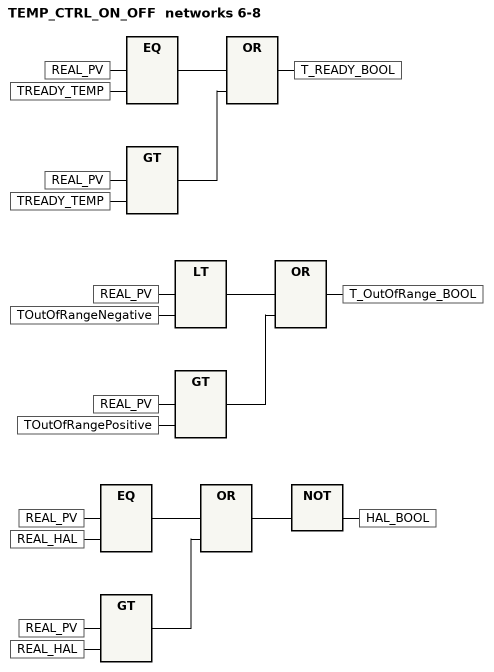
[picture p96: TEMP_CTRL_ON_OFF (FBD) networks 6-8]
_FBD_ (* Function Block Diagram *)
NETWORK 1
	DIV(INT_TO_REAL(TEMP_PV), 10) => REAL_PV
NETWORK 2
	T1:TON(IN: NOT ALWAYS_OFF, PT: T#100ms) => ALWAYS_ON_BOOL
NETWORK 3
	SUB(REAL_SV, REAL_T_READY) => TREADY_TEMP
NETWORK 4
	SUB(REAL_SV, REAL_HYS) => HYS_TEMP
NETWORK 5
	RS1:RS(SET: OR(AND(PLS1:R_TRIG(CLK: ALWAYS_ON_BOOL), LT(REAL_PV, REAL_SV)), OR(EQ(REAL_PV, HYS_TEMP), LT(REAL_PV, HYS_TEMP))), RESET1: OR(OR(EQ(REAL_PV, REAL_SV), GT(REAL_PV, REAL_SV)), NOT HAL_BOOL)) => OUT_BOOL
NETWORK 6
	OR(EQ(REAL_PV, TREADY_TEMP), GT(REAL_PV, TREADY_TEMP)) => T_READY_BOOL
NETWORK 7
	OR(LT(REAL_PV, TOutOfRangeNegative), GT(REAL_PV, TOutOfRangePositive)) => T_OutOfRange_BOOL
NETWORK 8
	NOT OR(EQ(REAL_PV, REAL_HAL), GT(REAL_PV, REAL_HAL)) => HAL_BOOL
_END_FBD_
(* the same logic as Structured Text *)
(* Network 1 *)
REAL_PV := INT_TO_REAL(TEMP_PV) / 10;
(* Network 2 *)
T1(IN := NOT ALWAYS_OFF, PT := T#100ms);
ALWAYS_ON_BOOL := T1.Q;
(* Network 3 *)
TREADY_TEMP := REAL_SV - REAL_T_READY;
(* Network 4 *)
HYS_TEMP := REAL_SV - REAL_HYS;
(* Network 5 *)
PLS1(CLK := ALWAYS_ON_BOOL);
RS1(SET := (PLS1.Q AND (REAL_PV < REAL_SV)) OR ((REAL_PV = HYS_TEMP) OR (REAL_PV < HYS_TEMP)), RESET1 := ((REAL_PV = REAL_SV) OR (REAL_PV > REAL_SV)) OR NOT HAL_BOOL);
OUT_BOOL := RS1.Q1;
(* Network 6 *)
T_READY_BOOL := (REAL_PV = TREADY_TEMP) OR (REAL_PV > TREADY_TEMP);
(* Network 7 *)
T_OutOfRange_BOOL := (REAL_PV < TOutOfRangeNegative) OR (REAL_PV > TOutOfRangePositive);
(* Network 8 *)
HAL_BOOL := NOT ((REAL_PV = REAL_HAL) OR (REAL_PV > REAL_HAL));
END_FUNCTION_BLOCK

(* POU TIMER_ALARM, LD *)
FUNCTION_BLOCK TIMER_ALARM
VAR_INPUT
	BOOL_SIGNAL_IN: BOOL;
	BOOL_ALMRST_PB: BOOL;
	BOOL_BZRST_PB: BOOL;
	INT_PV: INT;

END_VAR

VAR_OUTPUT
	ALM_MSG_BOOL: BOOL;
	BZ_OUT_BOOL: BOOL;
	EV_INT: INT;
END_VAR

VAR
	T1: TON;
	M0: BOOL;
	M1: BOOL;
	D200: TIME;
	D202: INT;
END_VAR
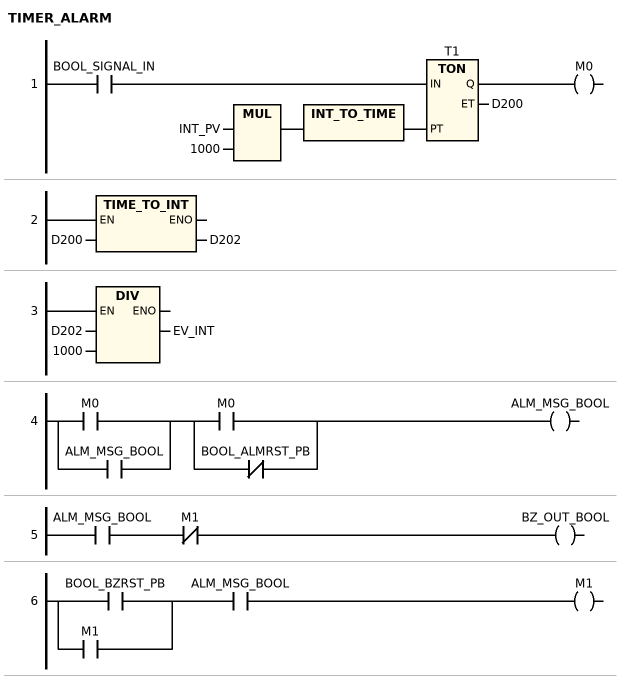
_LD_ (* Ladder Diagram *)
NETWORK 1
	[BOOL_SIGNAL_IN] - T1:TON(IN: *, PT: INT_TO_TIME(MUL(INT_PV, 1000)), ET => D200) --- (M0)
NETWORK 2
	*
		EN --- TIME_TO_INT(D200) => D202
NETWORK 3
	*
		EN --- DIV(D202, 1000) => EV_INT
NETWORK 4
	{ [M0] | [ALM_MSG_BOOL] } - { [M0] | [/BOOL_ALMRST_PB] } --- (ALM_MSG_BOOL)
NETWORK 5
	[ALM_MSG_BOOL] - [/M1] --- (BZ_OUT_BOOL)
NETWORK 6
	{ [BOOL_BZRST_PB] | [M1] } - [ALM_MSG_BOOL] --- (M1)
_END_LD_
(* the same logic as Structured Text *)
(* Network 1 *)
T1(IN := BOOL_SIGNAL_IN, PT := INT_TO_TIME(INT_PV * 1000));
D200 := T1.ET;
M0 := T1.Q;
(* Network 2 *)
D202 := TIME_TO_INT(D200);
(* Network 3 *)
EV_INT := D202 / 1000;
(* Network 4 *)
ALM_MSG_BOOL := (M0 OR ALM_MSG_BOOL) AND (M0 OR NOT BOOL_ALMRST_PB);
(* Network 5 *)
BZ_OUT_BOOL := ALM_MSG_BOOL AND NOT M1;
(* Network 6 *)
M1 := (BOOL_BZRST_PB OR M1) AND ALM_MSG_BOOL;
END_FUNCTION_BLOCK

(* POU TOWER_LIGHT, LD *)
FUNCTION_BLOCK TOWER_LIGHT
VAR_INPUT

	bAlarmOccur : BOOL;
	bMainOnOff : BOOL;
	bAutoStart : BOOL;
	bAutoProgress : BOOL;
	bAutoCycleStop: BOOL;
	bManualMode : BOOL;



END_VAR
VAR_OUTPUT
	bTowerLightRED : BOOL;
	bTowerLightYELLOW : BOOL;
	bTowerLightGREEN : BOOL;

END_VAR
VAR

	AlwaysOn : BOOL := TRUE;

	T1: TON;
	T2: TON;
END_VAR
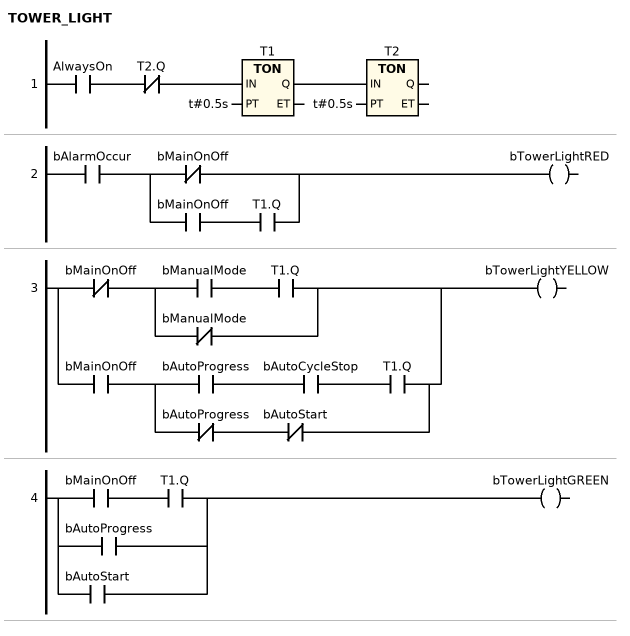
_LD_ (* Ladder Diagram *)
NETWORK 1
	[AlwaysOn] - [/T2.Q] - T1:TON(IN: *, PT: t#0.5s) - T2:TON(IN: *, PT: t#0.5s)
NETWORK 2
	[bAlarmOccur] - { [/bMainOnOff] | [bMainOnOff] - [T1.Q] } --- (bTowerLightRED)
NETWORK 3
	{ [/bMainOnOff] - { [bManualMode] - [T1.Q] | [/bManualMode] } | [bMainOnOff] - { [bAutoProgress] - [bAutoCycleStop] - [T1.Q] | [/bAutoProgress] - [/bAutoStart] } } --- (bTowerLightYELLOW)
NETWORK 4
	{ [bMainOnOff] - [T1.Q] | [bAutoProgress] | [bAutoStart] } --- (bTowerLightGREEN)
_END_LD_
(* the same logic as Structured Text *)
(* Network 1 *)
T1(IN := AlwaysOn AND NOT T2.Q, PT := t#0.5s);
T2(IN := T1.Q, PT := t#0.5s);
(* Network 2 *)
bTowerLightRED := bAlarmOccur AND (NOT bMainOnOff OR bMainOnOff AND T1.Q);
(* Network 3 *)
bTowerLightYELLOW := NOT bMainOnOff AND (bManualMode AND T1.Q OR NOT bManualMode) OR bMainOnOff AND (bAutoProgress AND bAutoCycleStop AND T1.Q OR NOT bAutoProgress AND NOT bAutoStart);
(* Network 4 *)
bTowerLightGREEN := bMainOnOff AND T1.Q OR bAutoProgress OR bAutoStart;
END_FUNCTION_BLOCK
